TYPE ST_AxisStatus :
STRUCT
    //Outputs & Status
    bAxisInitialized: BOOL := FALSE; //True when all parameters from actReadMcParameters are valid
    bAxisHasBeenRestored: BOOL := FALSE;
    bEnabled: BOOL; //Axis drive enabled
    bAxisReadyToMove: BOOL; //Axis enabled and input ok from additional equipment (e.g. airpad, brake).
    bCommandAborted: BOOL; //Command aborted output of the eCommand function blocks
    bBusy: BOOL; //Axis busy (eCommand function block is active)
    bDone: BOOL; //Last eCommand function block executed successfully
    //bDone will also be set with the InGear and InVelocity outputs
    //When InVelocity is set, fbMoveVelocity is still acitve, which is reflected by the bBusy status
    bInVelocity: BOOL; //MC_MoveVelocity has reached target velocity; will stay true until the movement stops
    bHomed: BOOL; //True when the axis has been successfully homed
    bMoving: BOOL; //Moving state from the NC
    bMovingForward: BOOL; //Moving forward indicator from NC
    bMovingBackward: BOOL; //Moving backward indicator from NC
    bInTargetPosition: BOOL; //True if the axis is in the target position
    bFwEnabled: BOOL; //Positive movement of axis is enabled/disabled
    bBwEnabled: BOOL; //Negative movement of axis is enabled/disabled
    bInterlockedFwd: BOOL; //True if the axis is interlocked in the forward direction
    bInterlockedBwd: BOOL; //True if the axis is interlocked in the backward direction
    bGeared: BOOL; //True if the axis is geared as a slave to another axis
    bBacklashCompensating: BOOL; //True if the axis is currently compensating for backlash
    bCoupledGear1: BOOL; //True if coupled to gear 1
    bCoupledGear2: BOOL; //True if coupled to gear 2
    bCoupledGear3: BOOL; //True if coupled to gear 3
    bCoupledGear4: BOOL; //True if coupled to gear 4
    bSlitsAxisBusy: BOOL; //True if an axis that belongs to the slits set is busy
    fActPosition: LREAL; //Actual position value
    fActTemperature: REAL; //Actual Temperature
    bHighTempAxisDisabled: BOOL := FALSE; //True if the axis is disabled due to high temperature
    bTempSensorError: BOOL; //Error when PT1OO is wrongly connected or disconnected
    nEncoderRawCounter AT %I*: UDINT; //Raw encoder counter value
    nStepperDriveCounter AT %I*: UDINT; //Raw internal counter value from the stepper drive
    fActVelocity: LREAL; //Current Velocity of the Axis
    bError: BOOL; //True if the axis is in an NC Error Stop state from Axis_Status
    nErrorID: UDINT; //ID of the last error from a motion function block or NC
    bSoEDriveDeviceError: BOOL; //SoE Drive hardware has an error (no warning)
    nSoEErrorID: UINT;
    nSoEDiagID: UDINT;
    bAirpadReady: BOOL; //True if airpad in ready to move state + feedback ok (if connected)
    bAirpadPressureError: BOOL; //True if pressure error
    bExternalBrakeReady: BOOL; //True if brake in ready to move state + feedback ok (if connected)
    bExternalBrakeFailure: BOOL; //True if brake engaged unexpectedly.
    bExternalBrakeTimeoutError: BOOL; //True if external brake id not report released in time
    bCommandHandlerMovePermit: BOOL; //True if CommandHandler has given permit to move
    bCommandHandlerReleasedMoveCmd: BOOL; //True if CommandHandler released the move command
    bCommandHandlerBufferingCommand: BOOL; //True if CommandHandler is waiting on a permit before releasing the command
    bCommandHandlerTimeoutError: BOOL; //True if CommandHandler did not receive a permit in time
    eInternalMotionCommand: E_MotionFunctions;
    stSwitchInfo: ST_SwitchInfo; //Trigger/Untrigger positions and values of switches
END_STRUCT
END_TYPE

(* stored: Version 1.1.0.1
   DUT ST_AxisStatus: Id {665afad4-438f-0e33-0727-6e8aec20b565} *)
